(* Logix 5000 project; controller ARS14002_PLC vendor 1 type 14 code 218 rev 30.11; software revision 30.01; part 13 of 13 *)
(* tags used below, declared in another part *)
   AN_1000A : CM_AI_SCL;
   AN_1000B : CM_AI_SCL;
   AN_101A : CM_AI_SCL;
   AN_101B : CM_AI_SCL;
   AN_101C : CM_AI_SCL;
   AN_200A : CM_AI_SCL;
   ARS_READY_TO_RECEIVE : BOOL;
   ARS_READY_TO_SEND : BOOL;
   ARS_TO_AT3 : UDT_IPC;
   CP_PID_MaxOut : REAL;
   EN_1250 : BOOL;   // HXR-1250 Enable Signal
   ESTOP_PL : CM_DO_GENERIC;
   ESTOP_TRIP : BOOL;
   EW_TEST_FIRSTSCAN : BOOL;
   EW_TEST_VFDSPD : BOOL;
   FCV_101A : CM_AO_VLV;
   FCV_101B : CM_AO_VLV;
   FCV_101C : CM_AO_VLV;
   FCV_102B : CM_AO_VLV;
   FCV_102C : CM_AO_VLV;
   FCV_204 : CM_AO_VLV;
   FIRST_SCAN_BIT : BOOL;
   FT_1002 : CM_AI_SCL;
   FT_202 : CM_AI_SCL;
   FVR800C_ChangeDir : BOOL;
   FVR800C_ChangeDirOnStop : BOOL;
   FVR800C_ClearFault_Reset_TMR : TIMER;
   FVR800C_RunHours : REAL;
   FVR800C_RunHoursCTU : COUNTER;
   FVR800C_RunTime : REAL;
   FVR800C_RunTime_CalcHigh : DINT;
   FVR800C_RunTime_CalcLow : DINT;
   FVR800C_RunTime_x100Hrs_Current : DINT;
   FVR800C_RunTimer : TIMER;
   FVR800D_ChangeDir : BOOL;
   FVR800D_ChangeDirOnStop : BOOL;
   FVR800D_ClearFault_Reset_TMR : TIMER;
   FVR800D_RunHours : REAL;
   FVR800D_RunHoursCTU : COUNTER;
   FVR800D_RunTime : REAL;
   FVR800D_RunTime_CalcHigh : DINT;
   FVR800D_RunTime_CalcLow : DINT;
   FVR800D_RunTime_x100Hrs_Current : DINT;
   FVR800D_RunTimer : TIMER;
   FVR_800C_RUNNING : BOOL;
   FVR_800C_ST : BOOL;
   FVR_800D_RUNNING : BOOL;
   FVR_800D_ST : BOOL;
   HXR_1250 : CM_DO_FVNR;
   MTR_200A : CM_DO_FVNR;
   MTR_550 : CM_DO_FVNR;
   P_800A_Direction : BOOL;
   P_800A_Direction_Toggle : BOOL;
   P_800A_RUN_OCCURRED : BOOL;
   P_800B_Direction : BOOL;
   P_800B_Direction_Toggle : BOOL;
   P_800B_RUN_OCCURRED : BOOL;
   P_800C : CM_DO_FVR;
   P_800C_Direction : BOOL;
   P_800C_Direction_Toggle : BOOL;
   P_800C_Fault : BOOL;
   P_800C_RUN_OCCURRED : BOOL;
   P_800D : CM_DO_FVR;
   P_800D_Direction : BOOL;
   P_800D_Direction_Toggle : BOOL;
   P_800D_Fault : BOOL;
   P_800D_RUN_OCCURRED : BOOL;
   PDT_1101A : CM_AI_SCL_ALT;
   PIDE_800 : PID_ENHANCED;
   PT_1003 : CM_AI_SCL;
   PT_101A : CM_AI_SCL;
   PT_101B : CM_AI_SCL;
   PT_101C : CM_AI_SCL;
   PT_902 : CM_AI_SCL;
   SV_1000 : CM_DO_GENERIC;
   SV_1000B : CM_DO_GENERIC;
   SV_1000C : CM_DO_GENERIC;
   SV_1000D : CM_DO_GENERIC;
   SV_1000E : CM_DO_GENERIC;
   SV_1001F : CM_DO_GENERIC;
   SV_1002F : CM_DO_GENERIC;
   SV_1005X : CM_DO_GENERIC;
   SV_101AF : CM_DO_GENERIC;
   SV_101AN : CM_DO_GENERIC;
   SV_101AP : CM_DO_GENERIC;
   SV_101BF : CM_DO_GENERIC;
   SV_101BN : CM_DO_GENERIC;
   SV_101BP : CM_DO_GENERIC;
   SV_101CF : CM_DO_GENERIC;
   SV_101CN : CM_DO_GENERIC;
   SV_101CP : CM_DO_GENERIC;
   SV_102AF : CM_DO_GENERIC;
   SV_102BF : CM_DO_GENERIC;
   SV_102CF : CM_DO_GENERIC;
   SV_1100P : CM_DO_GENERIC;
   SV_1104A : CM_DO_GENERIC;
   SV_1109AX : CM_DO_GENERIC;
   SV_1204 : CM_DO_GENERIC;
   SV_1206 : CM_DO_GENERIC;
   SV_1207X : CM_DO_GENERIC;
   SV_1208X : CM_DO_GENERIC;
   SV_1221F : CM_DO_GENERIC;
   SV_1251F : CM_DO_GENERIC;
   SV_1276 : CM_DO_GENERIC;
   SV_1304A : CM_DO_GENERIC;
   SV_1304B : CM_DO_GENERIC;
   SV_1309AX : CM_DO_GENERIC;
   SV_1309BX : CM_DO_GENERIC;
   SV_200A : CM_DO_GENERIC;
   SV_200B : CM_DO_GENERIC;
   SV_202F : CM_DO_GENERIC;
   SV_204F : CM_DO_GENERIC;
   SV_205 : CM_DO_GENERIC;
   SV_206 : CM_DO_GENERIC;
   SV_207F : CM_DO_GENERIC;
   SV_221X : CM_DO_GENERIC;
   SV_504F : CM_DO_GENERIC;
   SV_505X : CM_DO_GENERIC;
   SV_602A : CM_DO_GENERIC;
   SV_603F : CM_DO_GENERIC;
   SV_605F : CM_DO_GENERIC;
   SV_753F : CM_DO_GENERIC;
   SV_754F : CM_DO_GENERIC;
   SV_755F : CM_DO_GENERIC;
   SV_802AX : CM_DO_GENERIC;
   SV_802BX : CM_DO_GENERIC;
   SV_802CX : CM_DO_GENERIC;
   SV_802DX : CM_DO_GENERIC;
   TE_1003 : CM_AI_SCL;
   TimeStamp : DINT[7];
   VFD800A_ChangeDir : BOOL;
   VFD800A_ChangeDirOnStop : BOOL;
   VFD800A_ClearFault_Reset_TMR : TIMER;
   VFD800A_RunTime_CalcHigh : DINT;
   VFD800A_RunTime_CalcLow : DINT;
   VFD800A_RunTime_x100Hrs_Current : DINT;
   VFD800B_ChangeDir : BOOL;
   VFD800B_ChangeDirOnStop : BOOL;
   VFD800B_ClearFault_Reset_TMR : TIMER;
   VFD800B_RunTime_CalcHigh : DINT;
   VFD800B_RunTime_CalcLow : DINT;
   VFD800B_RunTime_x100Hrs_Current : DINT;
   VFD_800A_ST : BOOL;
   VFD_800B_ST : BOOL;
   WATCHDOG_OUT_100 : BOOL;
   WATCHDOG_OUT_1000 : BOOL;
   WATCHDOG_OUT_600 : BOOL;
   WATCHDOG_OUT_800 : BOOL;
   XV_1001 : CM_DO_VLV;
   XV_101B : CM_DO_VLV;
   XV_101C : CM_DO_VLV;
   XV_1123 : CM_DO_VLV;
   XV_1201 : CM_DO_VLV;
   XV_1202 : CM_DO_VLV;
   XV_1203 : CM_DO_VLV;
   XV_1204 : CM_DO_VLV;
   XV_1205 : CM_DO_VLV;
   XV_623 : CM_DO_VLV;
   XV_703 : CM_DO_VLV;
   XV_721A : CM_DO_VLV;
   XV_721B : CM_DO_VLV;
   XV_801A : CM_DO_VLV;
   XV_801B : CM_DO_VLV;
   XV_801C : CM_DO_VLV;
   XV_801D : CM_DO_VLV;
   XV_806 : CM_DO_VLV;
(* MainProgram, continued *)

ROUTINE _51_Outputs_VFD   (* ladder *)
// VFD output scaling and alarm handling routine
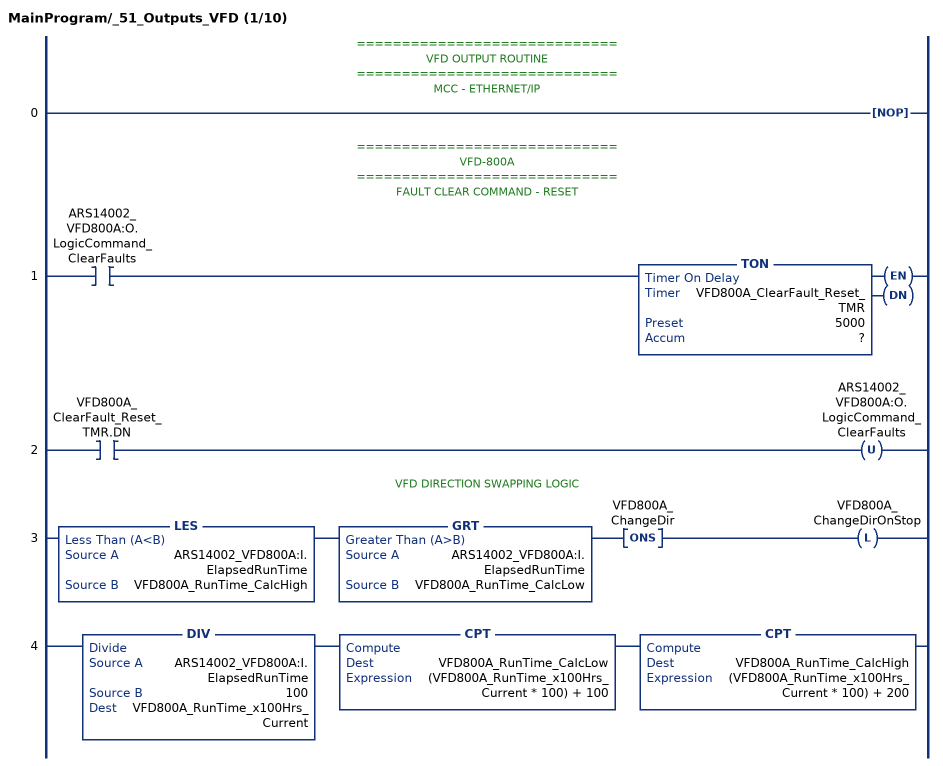
   // =============================
   // VFD OUTPUT ROUTINE
   // =============================
   // MCC - ETHERNET/IP
   0: NOP();
   // =============================
   // VFD-800A
   // =============================
   // FAULT CLEAR COMMAND - RESET
   1: XIC(ARS14002_VFD800A:O.LogicCommand_ClearFaults)TON(VFD800A_ClearFault_Reset_TMR,?,?);
   2: XIC(VFD800A_ClearFault_Reset_TMR.DN)OTU(ARS14002_VFD800A:O.LogicCommand_ClearFaults);
   // VFD DIRECTION SWAPPING LOGIC
   3: LES(ARS14002_VFD800A:I.ElapsedRunTime,VFD800A_RunTime_CalcHigh)GRT(ARS14002_VFD800A:I.ElapsedRunTime,VFD800A_RunTime_CalcLow)ONS(VFD800A_ChangeDir)OTL(VFD800A_ChangeDirOnStop);
   4: DIV(ARS14002_VFD800A:I.ElapsedRunTime,100,VFD800A_RunTime_x100Hrs_Current)CPT(VFD800A_RunTime_CalcLow,(VFD800A_RunTime_x100Hrs_Current * 100) + 100)CPT(VFD800A_RunTime_CalcHigh,(VFD800A_RunTime_x100Hrs_Current * 100) + 200);
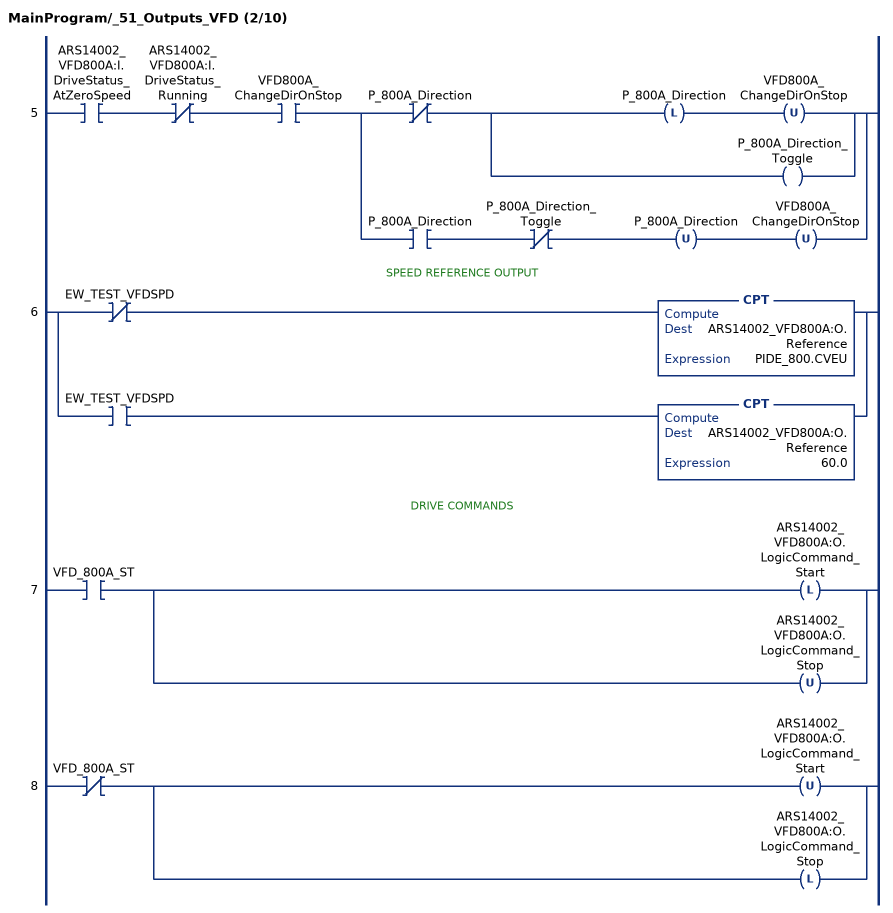
   5: XIC(ARS14002_VFD800A:I.DriveStatus_AtZeroSpeed)XIO(ARS14002_VFD800A:I.DriveStatus_Running)XIC(VFD800A_ChangeDirOnStop)[XIO(P_800A_Direction) [OTL(P_800A_Direction) OTU(VFD800A_ChangeDirOnStop) ,OTE(P_800A_Direction_Toggle) ] ,XIC(P_800A_Direction) XIO(P_800A_Direction_Toggle) OTU(P_800A_Direction) OTU(VFD800A_ChangeDirOnStop) ];
   // SPEED REFERENCE OUTPUT
   6: [XIO(EW_TEST_VFDSPD) CPT(ARS14002_VFD800A:O.Reference,PIDE_800.CVEU) ,XIC(EW_TEST_VFDSPD) CPT(ARS14002_VFD800A:O.Reference,60.0) ];
   // DRIVE COMMANDS
   7: XIC(VFD_800A_ST)[OTL(ARS14002_VFD800A:O.LogicCommand_Start) ,OTU(ARS14002_VFD800A:O.LogicCommand_Stop) ];
   8: XIO(VFD_800A_ST)[OTU(ARS14002_VFD800A:O.LogicCommand_Start) ,OTL(ARS14002_VFD800A:O.LogicCommand_Stop) ];
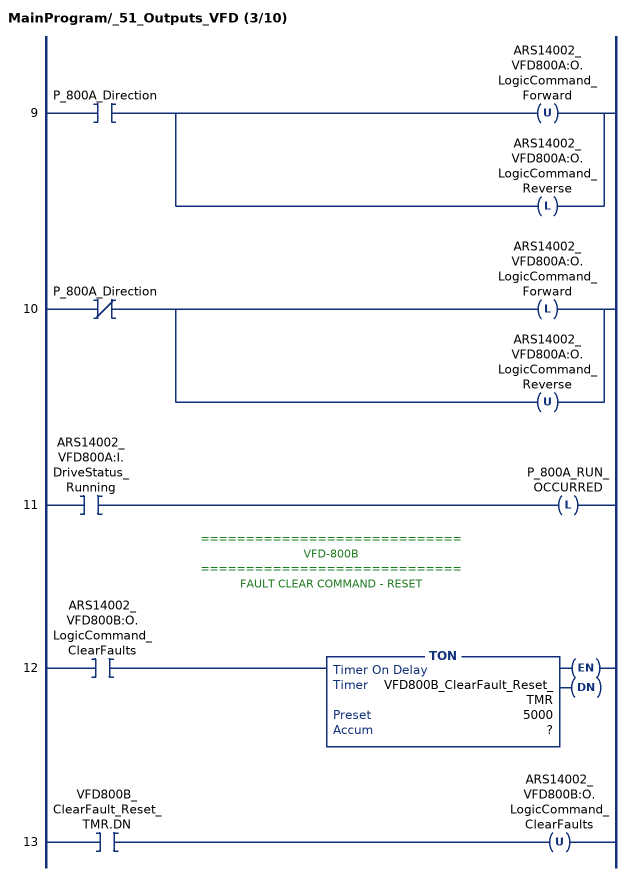
   9: XIC(P_800A_Direction)[OTU(ARS14002_VFD800A:O.LogicCommand_Forward) ,OTL(ARS14002_VFD800A:O.LogicCommand_Reverse) ];
   10: XIO(P_800A_Direction)[OTL(ARS14002_VFD800A:O.LogicCommand_Forward) ,OTU(ARS14002_VFD800A:O.LogicCommand_Reverse) ];
   11: XIC(ARS14002_VFD800A:I.DriveStatus_Running)OTL(P_800A_RUN_OCCURRED);
   // =============================
   // VFD-800B
   // =============================
   // FAULT CLEAR COMMAND - RESET
   12: XIC(ARS14002_VFD800B:O.LogicCommand_ClearFaults)TON(VFD800B_ClearFault_Reset_TMR,?,?);
   13: XIC(VFD800B_ClearFault_Reset_TMR.DN)OTU(ARS14002_VFD800B:O.LogicCommand_ClearFaults);
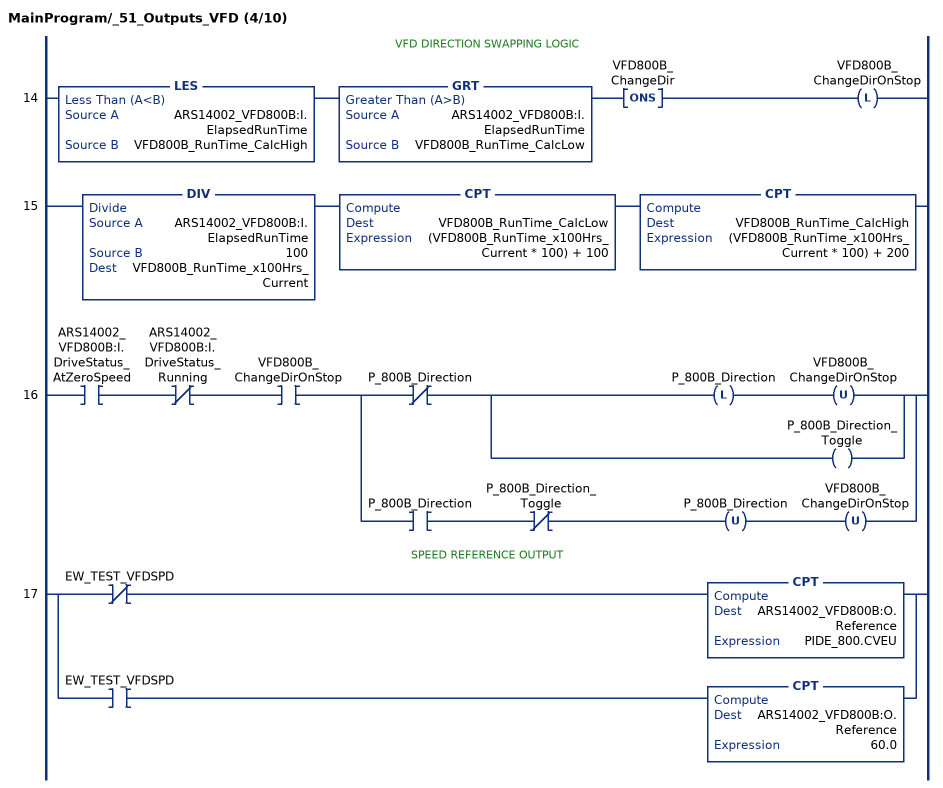
   // VFD DIRECTION SWAPPING LOGIC
   14: LES(ARS14002_VFD800B:I.ElapsedRunTime,VFD800B_RunTime_CalcHigh)GRT(ARS14002_VFD800B:I.ElapsedRunTime,VFD800B_RunTime_CalcLow)ONS(VFD800B_ChangeDir)OTL(VFD800B_ChangeDirOnStop);
   15: DIV(ARS14002_VFD800B:I.ElapsedRunTime,100,VFD800B_RunTime_x100Hrs_Current)CPT(VFD800B_RunTime_CalcLow,(VFD800B_RunTime_x100Hrs_Current * 100) + 100)CPT(VFD800B_RunTime_CalcHigh,(VFD800B_RunTime_x100Hrs_Current * 100) + 200);
   16: XIC(ARS14002_VFD800B:I.DriveStatus_AtZeroSpeed)XIO(ARS14002_VFD800B:I.DriveStatus_Running)XIC(VFD800B_ChangeDirOnStop)[XIO(P_800B_Direction) [OTL(P_800B_Direction) OTU(VFD800B_ChangeDirOnStop) ,OTE(P_800B_Direction_Toggle) ] ,XIC(P_800B_Direction) XIO(P_800B_Direction_Toggle) OTU(P_800B_Direction) OTU(VFD800B_ChangeDirOnStop) ];
   // SPEED REFERENCE OUTPUT
   17: [XIO(EW_TEST_VFDSPD) CPT(ARS14002_VFD800B:O.Reference,PIDE_800.CVEU) ,XIC(EW_TEST_VFDSPD) CPT(ARS14002_VFD800B:O.Reference,60.0) ];
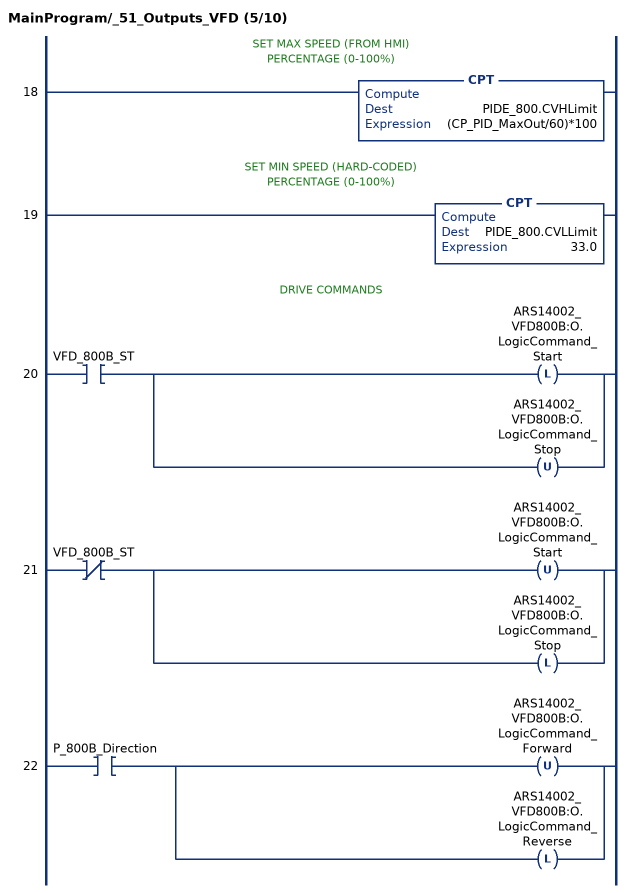
   // SET MAX SPEED (FROM HMI)
   // PERCENTAGE (0-100%)
   18: CPT(PIDE_800.CVHLimit,(CP_PID_MaxOut/60)*100);
   // SET MIN SPEED (HARD-CODED)
   // PERCENTAGE (0-100%)
   19: CPT(PIDE_800.CVLLimit,33.0);
   // DRIVE COMMANDS
   20: XIC(VFD_800B_ST)[OTL(ARS14002_VFD800B:O.LogicCommand_Start) ,OTU(ARS14002_VFD800B:O.LogicCommand_Stop) ];
   21: XIO(VFD_800B_ST)[OTU(ARS14002_VFD800B:O.LogicCommand_Start) ,OTL(ARS14002_VFD800B:O.LogicCommand_Stop) ];
   22: XIC(P_800B_Direction)[OTU(ARS14002_VFD800B:O.LogicCommand_Forward) ,OTL(ARS14002_VFD800B:O.LogicCommand_Reverse) ];
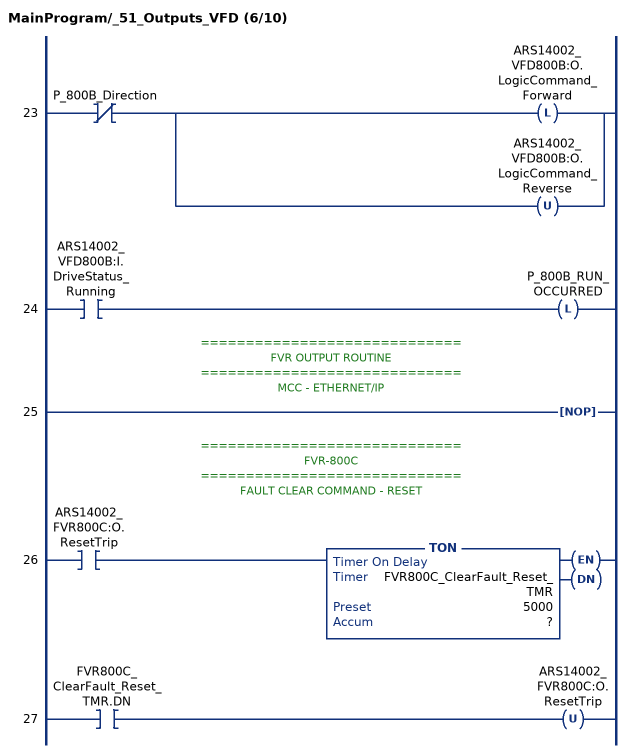
   23: XIO(P_800B_Direction)[OTL(ARS14002_VFD800B:O.LogicCommand_Forward) ,OTU(ARS14002_VFD800B:O.LogicCommand_Reverse) ];
   24: XIC(ARS14002_VFD800B:I.DriveStatus_Running)OTL(P_800B_RUN_OCCURRED);
   // =============================
   // FVR OUTPUT ROUTINE
   // =============================
   // MCC - ETHERNET/IP
   25: NOP();
   // =============================
   // FVR-800C
   // =============================
   // FAULT CLEAR COMMAND - RESET
   26: XIC(ARS14002_FVR800C:O.ResetTrip)TON(FVR800C_ClearFault_Reset_TMR,?,?);
   27: XIC(FVR800C_ClearFault_Reset_TMR.DN)OTU(ARS14002_FVR800C:O.ResetTrip);
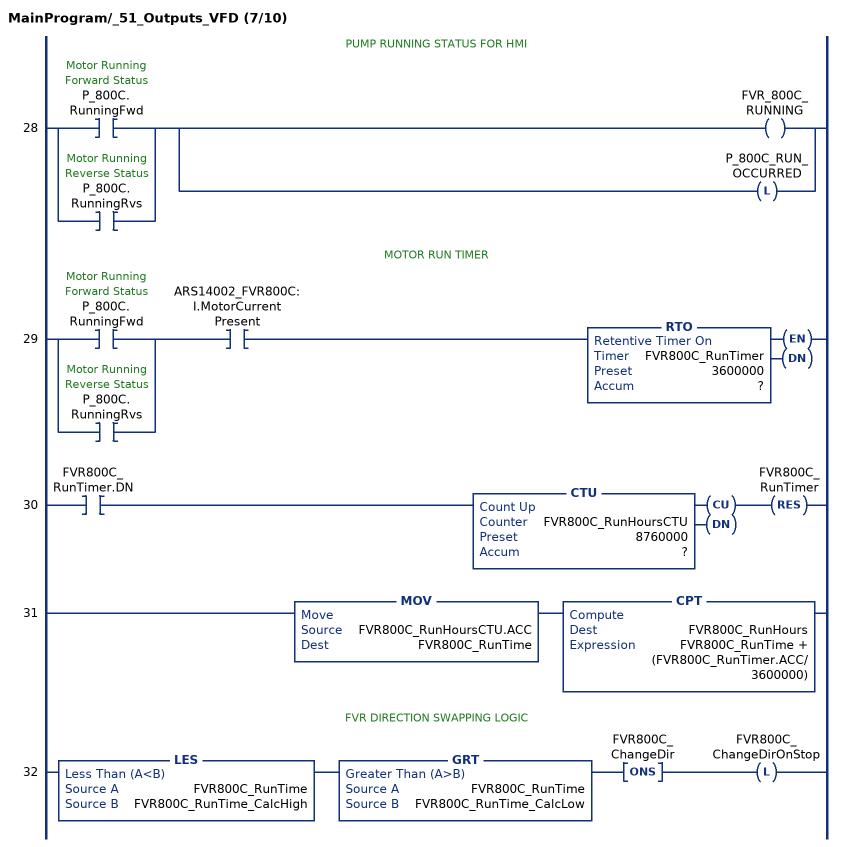
   // PUMP RUNNING STATUS FOR HMI
   28: [XIC(P_800C.RunningFwd) ,XIC(P_800C.RunningRvs) ][OTE(FVR_800C_RUNNING) ,OTL(P_800C_RUN_OCCURRED) ];
   // MOTOR RUN TIMER
   29: [XIC(P_800C.RunningFwd) ,XIC(P_800C.RunningRvs) ]XIC(ARS14002_FVR800C:I.MotorCurrentPresent)RTO(FVR800C_RunTimer,?,?);
   30: XIC(FVR800C_RunTimer.DN)CTU(FVR800C_RunHoursCTU,?,?)RES(FVR800C_RunTimer);
   31: MOV(FVR800C_RunHoursCTU.ACC,FVR800C_RunTime)CPT(FVR800C_RunHours,FVR800C_RunTime + (FVR800C_RunTimer.ACC/3600000));
   // FVR DIRECTION SWAPPING LOGIC
   32: LES(FVR800C_RunTime,FVR800C_RunTime_CalcHigh)GRT(FVR800C_RunTime,FVR800C_RunTime_CalcLow)ONS(FVR800C_ChangeDir)OTL(FVR800C_ChangeDirOnStop);
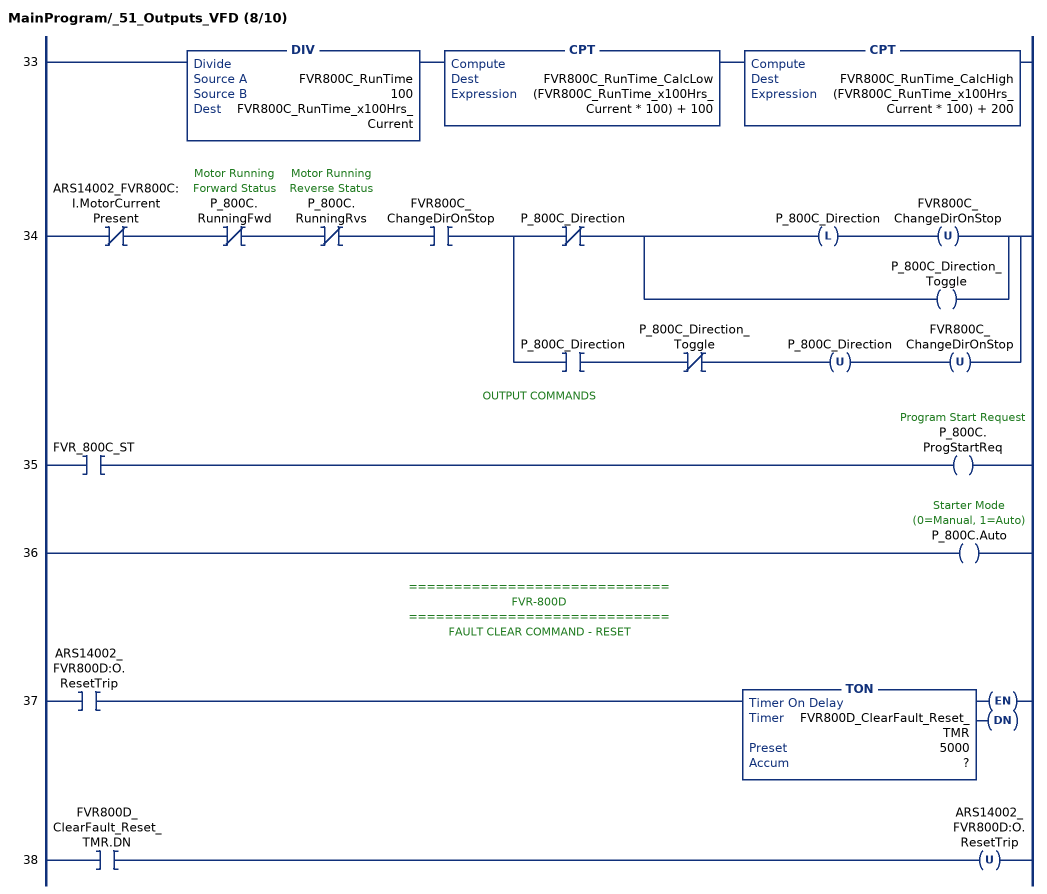
   33: DIV(FVR800C_RunTime,100,FVR800C_RunTime_x100Hrs_Current)CPT(FVR800C_RunTime_CalcLow,(FVR800C_RunTime_x100Hrs_Current * 100) + 100)CPT(FVR800C_RunTime_CalcHigh,(FVR800C_RunTime_x100Hrs_Current * 100) + 200);
   34: XIO(ARS14002_FVR800C:I.MotorCurrentPresent)XIO(P_800C.RunningFwd)XIO(P_800C.RunningRvs)XIC(FVR800C_ChangeDirOnStop)[XIO(P_800C_Direction) [OTL(P_800C_Direction) OTU(FVR800C_ChangeDirOnStop) ,OTE(P_800C_Direction_Toggle) ] ,XIC(P_800C_Direction) XIO(P_800C_Direction_Toggle) OTU(P_800C_Direction) OTU(FVR800C_ChangeDirOnStop) ];
   // OUTPUT COMMANDS
   35: XIC(FVR_800C_ST)OTE(P_800C.ProgStartReq);
   36: OTE(P_800C.Auto);
   // =============================
   // FVR-800D
   // =============================
   // FAULT CLEAR COMMAND - RESET
   37: XIC(ARS14002_FVR800D:O.ResetTrip)TON(FVR800D_ClearFault_Reset_TMR,?,?);
   38: XIC(FVR800D_ClearFault_Reset_TMR.DN)OTU(ARS14002_FVR800D:O.ResetTrip);
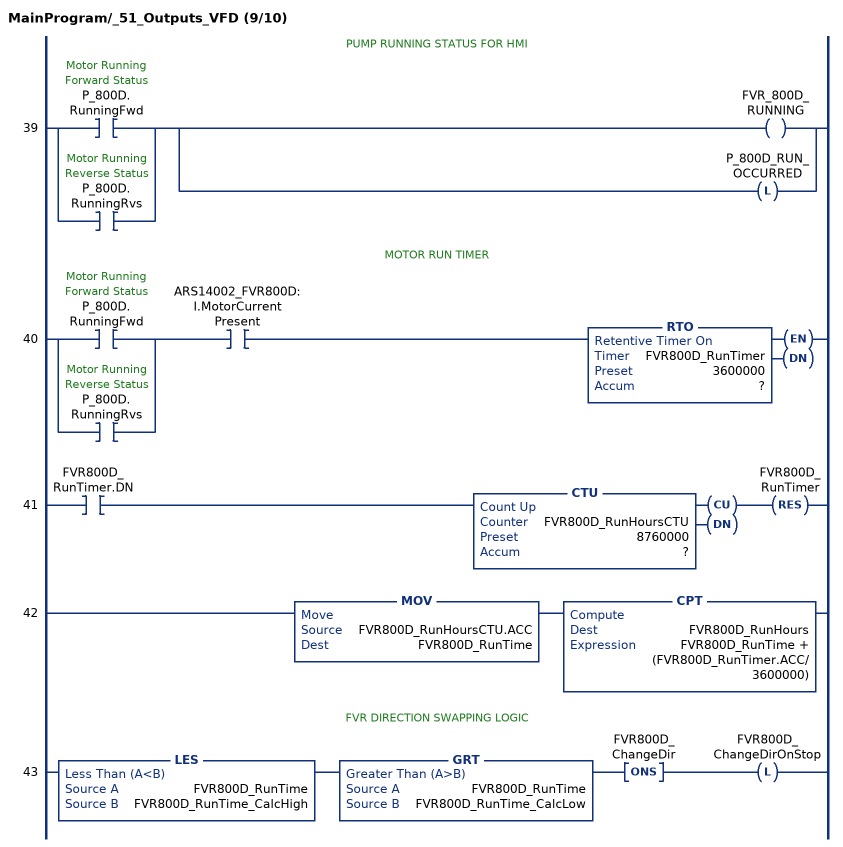
   // PUMP RUNNING STATUS FOR HMI
   39: [XIC(P_800D.RunningFwd) ,XIC(P_800D.RunningRvs) ][OTE(FVR_800D_RUNNING) ,OTL(P_800D_RUN_OCCURRED) ];
   // MOTOR RUN TIMER
   40: [XIC(P_800D.RunningFwd) ,XIC(P_800D.RunningRvs) ]XIC(ARS14002_FVR800D:I.MotorCurrentPresent)RTO(FVR800D_RunTimer,?,?);
   41: XIC(FVR800D_RunTimer.DN)CTU(FVR800D_RunHoursCTU,?,?)RES(FVR800D_RunTimer);
   42: MOV(FVR800D_RunHoursCTU.ACC,FVR800D_RunTime)CPT(FVR800D_RunHours,FVR800D_RunTime + (FVR800D_RunTimer.ACC/3600000));
   // FVR DIRECTION SWAPPING LOGIC
   43: LES(FVR800D_RunTime,FVR800D_RunTime_CalcHigh)GRT(FVR800D_RunTime,FVR800D_RunTime_CalcLow)ONS(FVR800D_ChangeDir)OTL(FVR800D_ChangeDirOnStop);
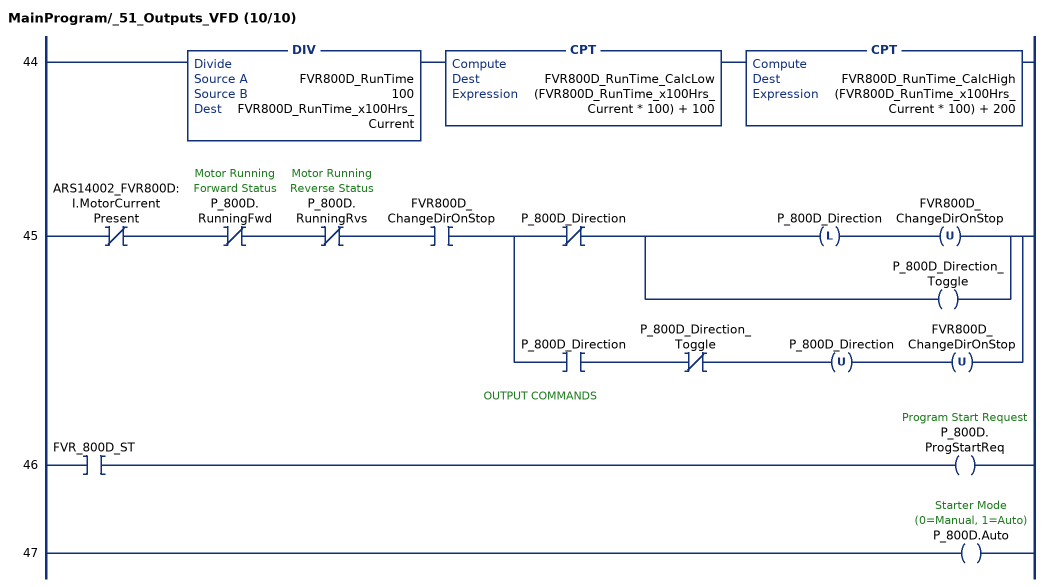
   44: DIV(FVR800D_RunTime,100,FVR800D_RunTime_x100Hrs_Current)CPT(FVR800D_RunTime_CalcLow,(FVR800D_RunTime_x100Hrs_Current * 100) + 100)CPT(FVR800D_RunTime_CalcHigh,(FVR800D_RunTime_x100Hrs_Current * 100) + 200);
   45: XIO(ARS14002_FVR800D:I.MotorCurrentPresent)XIO(P_800D.RunningFwd)XIO(P_800D.RunningRvs)XIC(FVR800D_ChangeDirOnStop)[XIO(P_800D_Direction) [OTL(P_800D_Direction) OTU(FVR800D_ChangeDirOnStop) ,OTE(P_800D_Direction_Toggle) ] ,XIC(P_800D_Direction) XIO(P_800D_Direction_Toggle) OTU(P_800D_Direction) OTU(FVR800D_ChangeDirOnStop) ];
   // OUTPUT COMMANDS
   46: XIC(FVR_800D_ST)OTE(P_800D.ProgStartReq);
   47: OTE(P_800D.Auto);
END_ROUTINE

ROUTINE _52_Outputs_Discrete   (* ladder *)
// On/Off Output process control and alarm handling
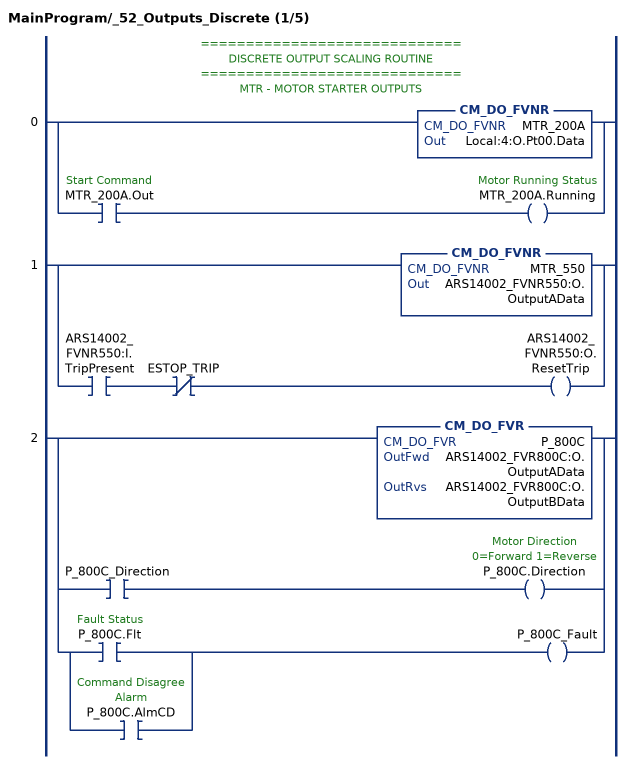
   // =============================
   // DISCRETE OUTPUT SCALING ROUTINE
   // =============================
   // MTR - MOTOR STARTER OUTPUTS
   0: [CM_DO_FVNR(MTR_200A,Local:4:O.Pt00.Data) ,XIC(MTR_200A.Out) OTE(MTR_200A.Running) ];
   1: [CM_DO_FVNR(MTR_550,ARS14002_FVNR550:O.OutputAData) ,XIC(ARS14002_FVNR550:I.TripPresent) XIO(ESTOP_TRIP) OTE(ARS14002_FVNR550:O.ResetTrip) ];
   2: [CM_DO_FVR(P_800C,ARS14002_FVR800C:O.OutputAData,ARS14002_FVR800C:O.OutputBData) ,[XIC(P_800C_Direction) OTE(P_800C.Direction) ,[XIC(P_800C.Flt) ,XIC(P_800C.AlmCD) ] OTE(P_800C_Fault) ] ];
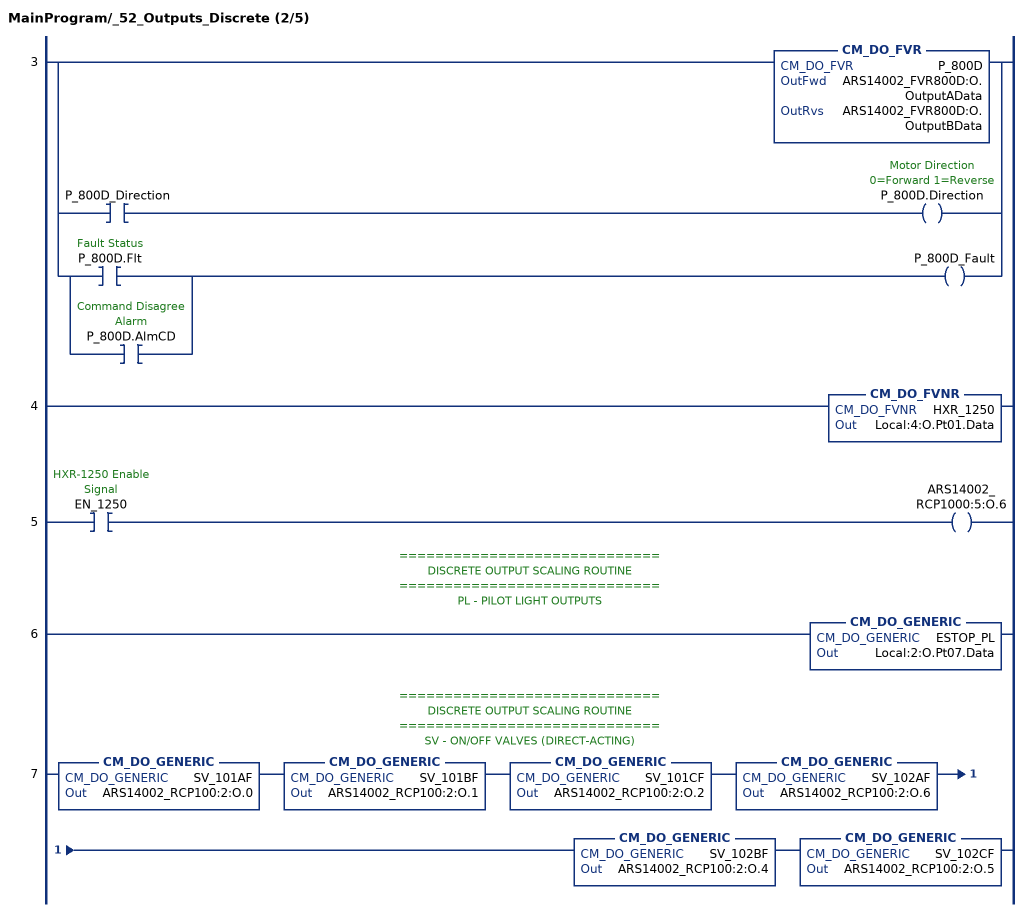
   3: [CM_DO_FVR(P_800D,ARS14002_FVR800D:O.OutputAData,ARS14002_FVR800D:O.OutputBData) ,[XIC(P_800D_Direction) OTE(P_800D.Direction) ,[XIC(P_800D.Flt) ,XIC(P_800D.AlmCD) ] OTE(P_800D_Fault) ] ];
   4: CM_DO_FVNR(HXR_1250,Local:4:O.Pt01.Data);
   5: XIC(EN_1250)OTE(ARS14002_RCP1000:5:O.6);
   // =============================
   // DISCRETE OUTPUT SCALING ROUTINE
   // =============================
   // PL - PILOT LIGHT OUTPUTS
   6: CM_DO_GENERIC(ESTOP_PL,Local:2:O.Pt07.Data);
   // =============================
   // DISCRETE OUTPUT SCALING ROUTINE
   // =============================
   // SV - ON/OFF VALVES (DIRECT-ACTING)
   7: CM_DO_GENERIC(SV_101AF,ARS14002_RCP100:2:O.0)CM_DO_GENERIC(SV_101BF,ARS14002_RCP100:2:O.1)CM_DO_GENERIC(SV_101CF,ARS14002_RCP100:2:O.2)CM_DO_GENERIC(SV_102AF,ARS14002_RCP100:2:O.6)CM_DO_GENERIC(SV_102BF,ARS14002_RCP100:2:O.4)CM_DO_GENERIC(SV_102CF,ARS14002_RCP100:2:O.5);
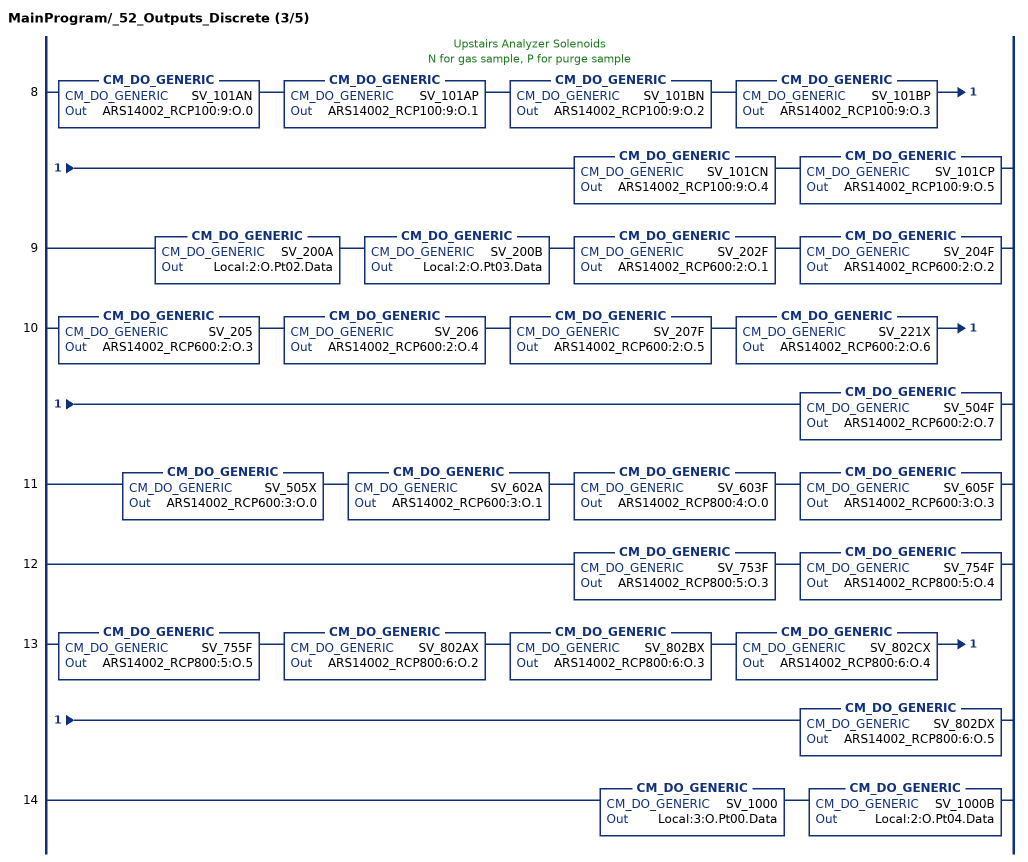
   // Upstairs Analyzer Solenoids
   // N for gas sample, P for purge sample
   8: CM_DO_GENERIC(SV_101AN,ARS14002_RCP100:9:O.0)CM_DO_GENERIC(SV_101AP,ARS14002_RCP100:9:O.1)CM_DO_GENERIC(SV_101BN,ARS14002_RCP100:9:O.2)CM_DO_GENERIC(SV_101BP,ARS14002_RCP100:9:O.3)CM_DO_GENERIC(SV_101CN,ARS14002_RCP100:9:O.4)CM_DO_GENERIC(SV_101CP,ARS14002_RCP100:9:O.5);
   9: CM_DO_GENERIC(SV_200A,Local:2:O.Pt02.Data)CM_DO_GENERIC(SV_200B,Local:2:O.Pt03.Data)CM_DO_GENERIC(SV_202F,ARS14002_RCP600:2:O.1)CM_DO_GENERIC(SV_204F,ARS14002_RCP600:2:O.2);
   10: CM_DO_GENERIC(SV_205,ARS14002_RCP600:2:O.3)CM_DO_GENERIC(SV_206,ARS14002_RCP600:2:O.4)CM_DO_GENERIC(SV_207F,ARS14002_RCP600:2:O.5)CM_DO_GENERIC(SV_221X,ARS14002_RCP600:2:O.6)CM_DO_GENERIC(SV_504F,ARS14002_RCP600:2:O.7);
   11: CM_DO_GENERIC(SV_505X,ARS14002_RCP600:3:O.0)CM_DO_GENERIC(SV_602A,ARS14002_RCP600:3:O.1)CM_DO_GENERIC(SV_603F,ARS14002_RCP800:4:O.0)CM_DO_GENERIC(SV_605F,ARS14002_RCP600:3:O.3);
   12: CM_DO_GENERIC(SV_753F,ARS14002_RCP800:5:O.3)CM_DO_GENERIC(SV_754F,ARS14002_RCP800:5:O.4);
   13: CM_DO_GENERIC(SV_755F,ARS14002_RCP800:5:O.5)CM_DO_GENERIC(SV_802AX,ARS14002_RCP800:6:O.2)CM_DO_GENERIC(SV_802BX,ARS14002_RCP800:6:O.3)CM_DO_GENERIC(SV_802CX,ARS14002_RCP800:6:O.4)CM_DO_GENERIC(SV_802DX,ARS14002_RCP800:6:O.5);
   14: CM_DO_GENERIC(SV_1000,Local:3:O.Pt00.Data)CM_DO_GENERIC(SV_1000B,Local:2:O.Pt04.Data);
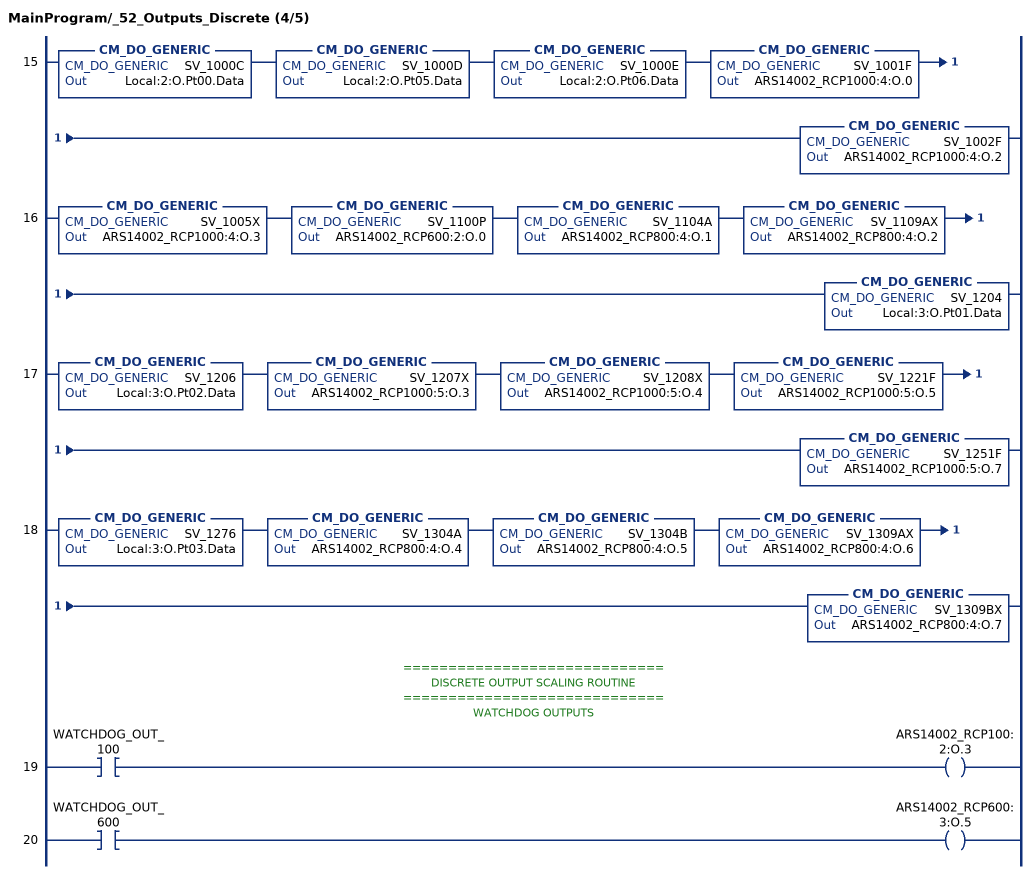
   15: CM_DO_GENERIC(SV_1000C,Local:2:O.Pt00.Data)CM_DO_GENERIC(SV_1000D,Local:2:O.Pt05.Data)CM_DO_GENERIC(SV_1000E,Local:2:O.Pt06.Data)CM_DO_GENERIC(SV_1001F,ARS14002_RCP1000:4:O.0)CM_DO_GENERIC(SV_1002F,ARS14002_RCP1000:4:O.2);
   16: CM_DO_GENERIC(SV_1005X,ARS14002_RCP1000:4:O.3)CM_DO_GENERIC(SV_1100P,ARS14002_RCP600:2:O.0)CM_DO_GENERIC(SV_1104A,ARS14002_RCP800:4:O.1)CM_DO_GENERIC(SV_1109AX,ARS14002_RCP800:4:O.2)CM_DO_GENERIC(SV_1204,Local:3:O.Pt01.Data);
   17: CM_DO_GENERIC(SV_1206,Local:3:O.Pt02.Data)CM_DO_GENERIC(SV_1207X,ARS14002_RCP1000:5:O.3)CM_DO_GENERIC(SV_1208X,ARS14002_RCP1000:5:O.4)CM_DO_GENERIC(SV_1221F,ARS14002_RCP1000:5:O.5)CM_DO_GENERIC(SV_1251F,ARS14002_RCP1000:5:O.7);
   18: CM_DO_GENERIC(SV_1276,Local:3:O.Pt03.Data)CM_DO_GENERIC(SV_1304A,ARS14002_RCP800:4:O.4)CM_DO_GENERIC(SV_1304B,ARS14002_RCP800:4:O.5)CM_DO_GENERIC(SV_1309AX,ARS14002_RCP800:4:O.6)CM_DO_GENERIC(SV_1309BX,ARS14002_RCP800:4:O.7);
   // =============================
   // DISCRETE OUTPUT SCALING ROUTINE
   // =============================
   // WATCHDOG OUTPUTS
   19: XIC(WATCHDOG_OUT_100)OTE(ARS14002_RCP100:2:O.3);
   20: XIC(WATCHDOG_OUT_600)OTE(ARS14002_RCP600:3:O.5);
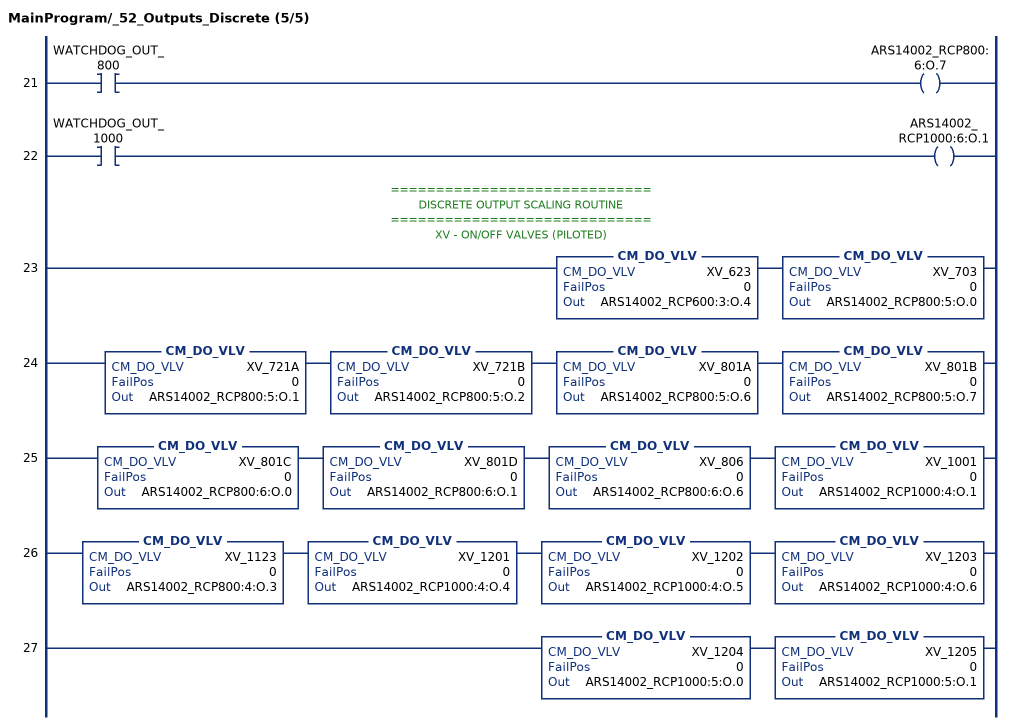
   21: XIC(WATCHDOG_OUT_800)OTE(ARS14002_RCP800:6:O.7);
   22: XIC(WATCHDOG_OUT_1000)OTE(ARS14002_RCP1000:6:O.1);
   // =============================
   // DISCRETE OUTPUT SCALING ROUTINE
   // =============================
   // XV - ON/OFF VALVES (PILOTED)
   23: CM_DO_VLV(XV_623,0,ARS14002_RCP600:3:O.4)CM_DO_VLV(XV_703,0,ARS14002_RCP800:5:O.0);
   24: CM_DO_VLV(XV_721A,0,ARS14002_RCP800:5:O.1)CM_DO_VLV(XV_721B,0,ARS14002_RCP800:5:O.2)CM_DO_VLV(XV_801A,0,ARS14002_RCP800:5:O.6)CM_DO_VLV(XV_801B,0,ARS14002_RCP800:5:O.7);
   25: CM_DO_VLV(XV_801C,0,ARS14002_RCP800:6:O.0)CM_DO_VLV(XV_801D,0,ARS14002_RCP800:6:O.1)CM_DO_VLV(XV_806,0,ARS14002_RCP800:6:O.6)CM_DO_VLV(XV_1001,0,ARS14002_RCP1000:4:O.1);
   26: CM_DO_VLV(XV_1123,0,ARS14002_RCP800:4:O.3)CM_DO_VLV(XV_1201,0,ARS14002_RCP1000:4:O.4)CM_DO_VLV(XV_1202,0,ARS14002_RCP1000:4:O.5)CM_DO_VLV(XV_1203,0,ARS14002_RCP1000:4:O.6);
   27: CM_DO_VLV(XV_1204,0,ARS14002_RCP1000:5:O.0)CM_DO_VLV(XV_1205,0,ARS14002_RCP1000:5:O.1);
END_ROUTINE

ROUTINE _53_Outputs_IPC   (* ladder *)
// Output Mapping Routine
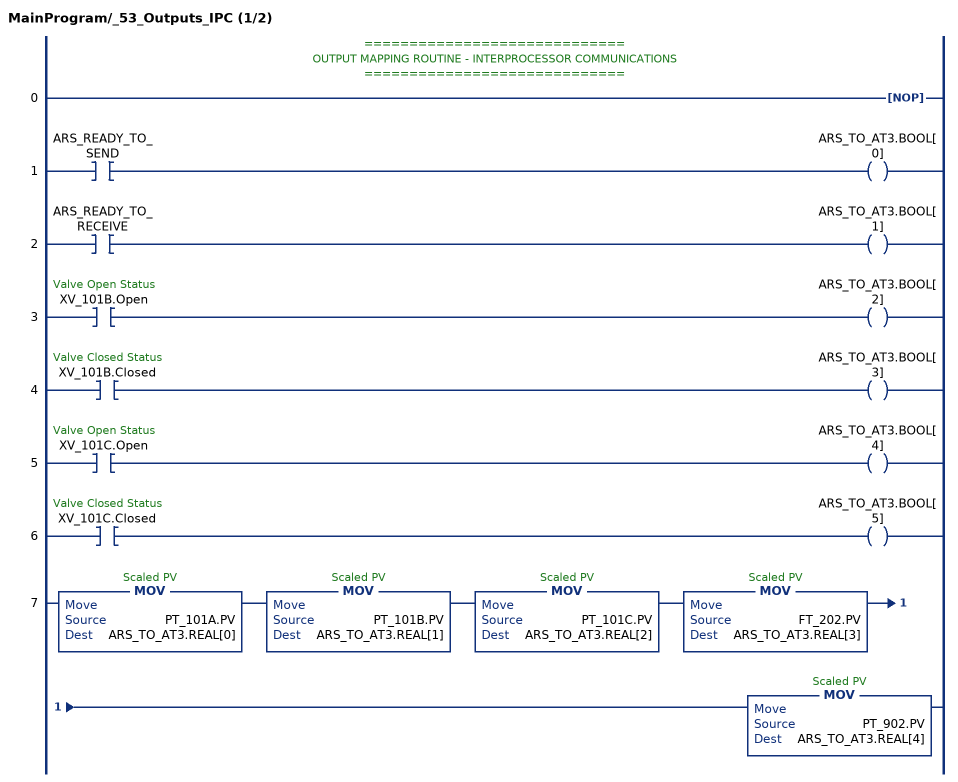
   // =============================
   // OUTPUT MAPPING ROUTINE - INTERPROCESSOR COMMUNICATIONS
   // =============================
   0: NOP();
   1: XIC(ARS_READY_TO_SEND)OTE(ARS_TO_AT3.BOOL[0]);
   2: XIC(ARS_READY_TO_RECEIVE)OTE(ARS_TO_AT3.BOOL[1]);
   3: XIC(XV_101B.Open)OTE(ARS_TO_AT3.BOOL[2]);
   4: XIC(XV_101B.Closed)OTE(ARS_TO_AT3.BOOL[3]);
   5: XIC(XV_101C.Open)OTE(ARS_TO_AT3.BOOL[4]);
   6: XIC(XV_101C.Closed)OTE(ARS_TO_AT3.BOOL[5]);
   7: MOV(PT_101A.PV,ARS_TO_AT3.REAL[0])MOV(PT_101B.PV,ARS_TO_AT3.REAL[1])MOV(PT_101C.PV,ARS_TO_AT3.REAL[2])MOV(FT_202.PV,ARS_TO_AT3.REAL[3])MOV(PT_902.PV,ARS_TO_AT3.REAL[4]);
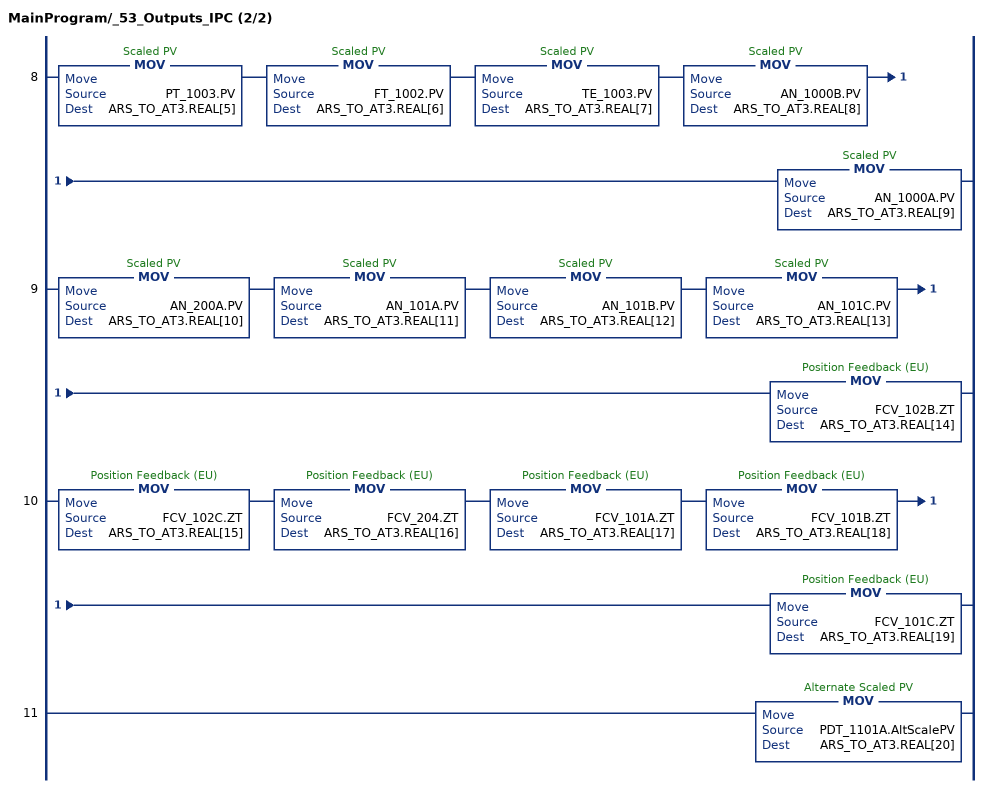
   8: MOV(PT_1003.PV,ARS_TO_AT3.REAL[5])MOV(FT_1002.PV,ARS_TO_AT3.REAL[6])MOV(TE_1003.PV,ARS_TO_AT3.REAL[7])MOV(AN_1000B.PV,ARS_TO_AT3.REAL[8])MOV(AN_1000A.PV,ARS_TO_AT3.REAL[9]);
   9: MOV(AN_200A.PV,ARS_TO_AT3.REAL[10])MOV(AN_101A.PV,ARS_TO_AT3.REAL[11])MOV(AN_101B.PV,ARS_TO_AT3.REAL[12])MOV(AN_101C.PV,ARS_TO_AT3.REAL[13])MOV(FCV_102B.ZT,ARS_TO_AT3.REAL[14]);
   10: MOV(FCV_102C.ZT,ARS_TO_AT3.REAL[15])MOV(FCV_204.ZT,ARS_TO_AT3.REAL[16])MOV(FCV_101A.ZT,ARS_TO_AT3.REAL[17])MOV(FCV_101B.ZT,ARS_TO_AT3.REAL[18])MOV(FCV_101C.ZT,ARS_TO_AT3.REAL[19]);
   11: MOV(PDT_1101A.AltScalePV,ARS_TO_AT3.REAL[20]);
END_ROUTINE

ROUTINE MainRoutine   (* ladder *)
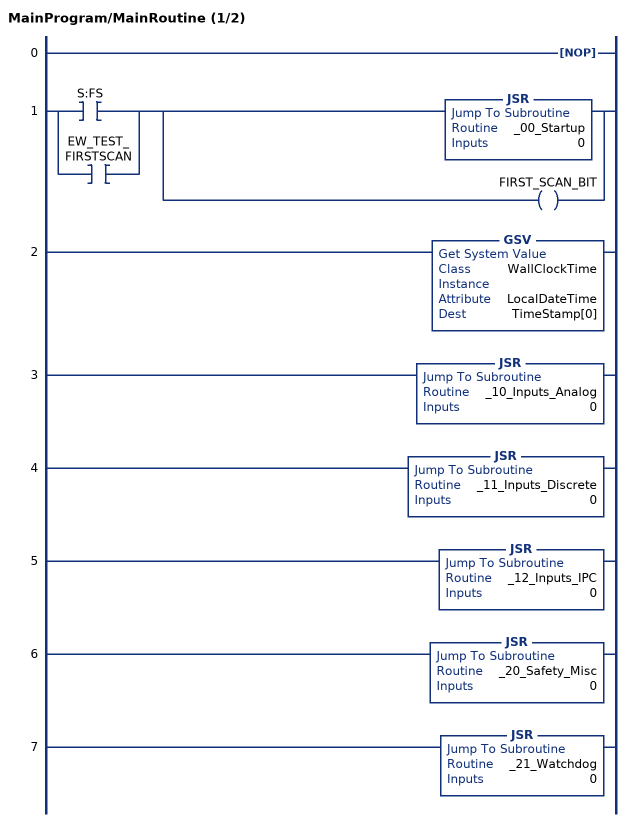
   0: NOP();
   1: [XIC(S:FS) ,XIC(EW_TEST_FIRSTSCAN) ][JSR(_00_Startup,0) ,OTE(FIRST_SCAN_BIT) ];
   2: GSV(WallClockTime,,LocalDateTime,TimeStamp[0]);
   3: JSR(_10_Inputs_Analog,0);
   4: JSR(_11_Inputs_Discrete,0);
   5: JSR(_12_Inputs_IPC,0);
   6: JSR(_20_Safety_Misc,0);
   7: JSR(_21_Watchdog,0);
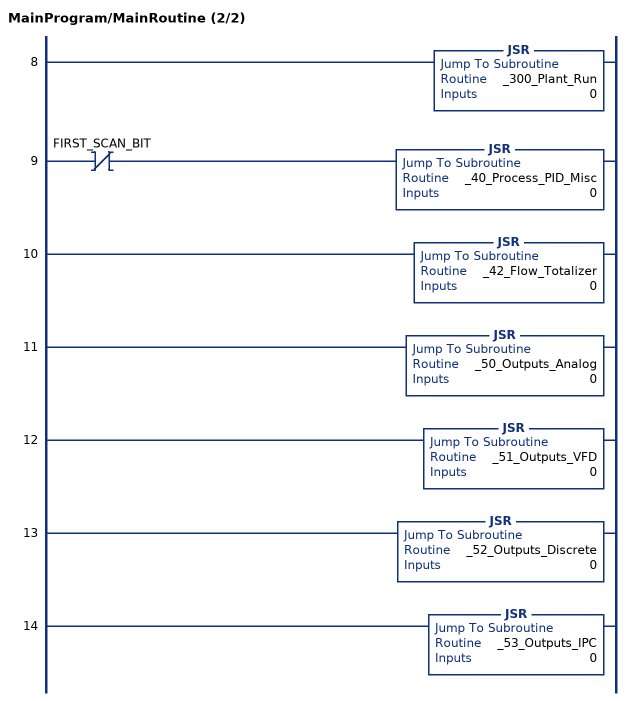
   8: JSR(_300_Plant_Run,0);
   9: XIO(FIRST_SCAN_BIT)JSR(_40_Process_PID_Misc,0);
   10: JSR(_42_Flow_Totalizer,0);
   11: JSR(_50_Outputs_Analog,0);
   12: JSR(_51_Outputs_VFD,0);
   13: JSR(_52_Outputs_Discrete,0);
   14: JSR(_53_Outputs_IPC,0);
END_ROUTINE
END_PROGRAM
